
FUNCTION CB_ge_tod : BOOL


TITLE = ' Test Whether IN0 is greater than or equal to IN1 '
VERSION : '1.0'
AUTHOR  : CB
NAME    : ge_tod
FAMILY  : TNI

VAR_INPUT
    IN0 : TOD;
    IN1 : TOD;
END_VAR

BEGIN

CB_ge_tod := (IN0 >= IN1);

END_FUNCTION
